// TIA Portal V19 export
TYPE "LAF_typeAxisProductionParameters"
// stored: Access Published
   STRUCT
      upperVel : LReal := 500.0;   // 产品模式速度上限
      distanceList : Array[0..99] of "LAF_typeAxisMotionParameters";
   END_STRUCT;
END_TYPE
